// SIMATIC S7-200 project (STEP 7-Micro/WIN), CPU 221 REL 01.10

ORGANIZATION_BLOCK PRINCIPAL:OB1
TITLE=EJERCICIO 3 BOTONES 3 FOCOS
BEGIN
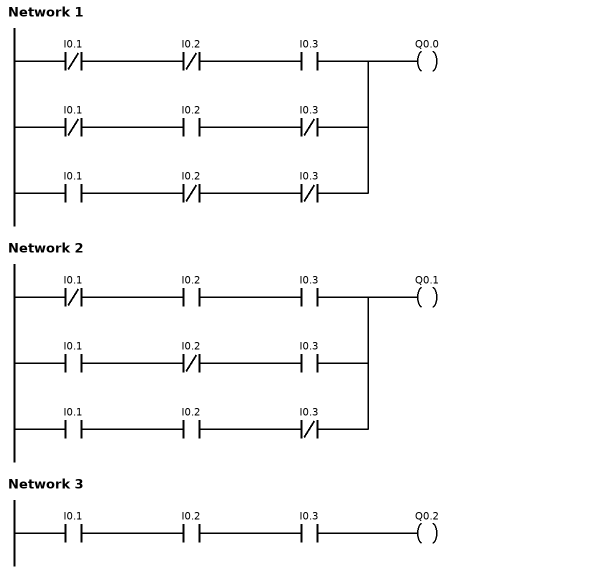
Network 1
LDN    I0.1
AN     I0.2
A      I0.3
LDN    I0.1
A      I0.2
AN     I0.3
OLD
LD     I0.1
AN     I0.2
AN     I0.3
OLD
=      Q0.0
Network 2
LDN    I0.1
A      I0.2
A      I0.3
LD     I0.1
AN     I0.2
A      I0.3
OLD
LD     I0.1
A      I0.2
AN     I0.3
OLD
=      Q0.1
Network 3
LD     I0.1
A      I0.2
A      I0.3
=      Q0.2
END_ORGANIZATION_BLOCK
